TYPE TFCentratoreManCmd :
STRUCT
	Ax : TFAxCentratoreManCmd;
	ResetModulo : bool;	
END_STRUCT
END_TYPE

(* stored: Version 1.1.0.1, ProductVersion 3.1.4024.11
   DUT TFCentratoreManCmd: Id {2bb084e1-b35c-4358-8321-eaf252d26a32} *)
